// Created by Dimitar Stojanov 06.2023 

//Functionality: Use this block to scale Analog Outputs

FUNCTION_BLOCK FB_AnalogOutput
VAR_INPUT
	i_rValue 							:REAL;
	i_rData_Low 						:REAL;
	i_rData_High 						:REAL;
	i_rScaled_Low						:INT	:=0;
	i_rScaled_High						:INT	:=32676;
	i_iOffset 							:INT;
	
END_VAR
VAR_OUTPUT
	q_iScaled							:INT;
END_VAR
VAR
	K								    :REAL;
END_VAR

K := ((i_rScaled_High - i_rScaled_Low) / (i_rData_High - i_rData_Low));
q_iScaled:=REAL_TO_INT((K * i_rValue) + i_iOffset);

END_FUNCTION_BLOCK

(* stored: Version 1.1.0.1, ProductVersion 3.1.4024.12
   POU FB_AnalogOutput: Id {cd9f5c74-7e84-4725-849e-005640f61686}, SpecialFunc None *)
